FUNCTION_BLOCK FB_GetByte_Test EXTENDS TcUnit.FB_TestSuite

TestGetLByte('Get LByte_1', nData := 16#1234, nExpected:= 16#34);
TestGetLByte('Get LByte_2', nData := 16#4321, nExpected:= 16#21);

TestGetHByte('Get HByte_1', nData := 16#1234, nExpected:= 16#12);
TestGetHByte('Get HByte_2', nData := 16#4321, nExpected:= 16#43);

METHOD TestGetHByte
VAR_INPUT
	sName : T_MaxString;	
	nData 	: WORD;
	nExpected : BYTE;
END_VAR

VAR		
	nResult : BYTE;
END_VAR
TEST(sName);


nResult := F_GetHByte(nData);
AssertEquals(Expected := nExpected,
             Actual := nResult,
             Message := 'Result value is not correct');	
	 
TEST_FINISHED();
END_METHOD

METHOD TestGetLByte
VAR_INPUT
	sName : T_MaxString;	
	nData 	: WORD;
	nExpected : BYTE;
END_VAR

VAR		
	nResult : BYTE;
END_VAR
TEST(sName);


nResult := F_GetLByte(nData);
AssertEquals(Expected := nExpected,
             Actual := nResult,
             Message := 'Result value is not correct');	
	 
TEST_FINISHED();
END_METHOD

END_FUNCTION_BLOCK

(* stored: Version 1.1.0.1, ProductVersion 3.1.4024.12
   POU FB_GetByte_Test: Id {58e66381-f177-0e77-3f12-b0b528107cbf}, SpecialFunc None
   Method TestGetHByte: Id {0fbec337-a69c-0cdc-16bc-300df263bb7b}
   Method TestGetLByte: Id {115390ec-8a7e-05c8-33f5-9cd305b2b06a} *)
